// Mitsubishi GX Works2 project: PLC_GROUP15   PLC: FX3G

// global labels: Global1
VAR_GLOBAL
  startDay AT X007 : BOOL;
  stayOn AT Y007 : BOOL;
  analogOutput AT D8282 : INT;
  checkStock AT M1 : BOOL;
  theDayEnd AT M20 : BOOL;
  validStock AT M2 : BOOL;
  lifeDay AT Y007 : BOOL;
  helpDayStart AT M22 : BOOL;
  petelInput AT D1100 : REAL;
END_VAR
VAR_GLOBAL CONSTANT
  petelMin : REAL := 280;
END_VAR
VAR_GLOBAL
  limonInput AT D1200 : REAL;
END_VAR
VAR_GLOBAL CONSTANT
  limonMin : REAL := 455;
END_VAR
VAR_GLOBAL
  meiatzevInput AT D1300 : REAL;
END_VAR
VAR_GLOBAL CONSTANT
  meiatzevMin : REAL := 105;
END_VAR
VAR_GLOBAL
  gummiInput AT D1400 : REAL;
END_VAR
VAR_GLOBAL CONSTANT
  gummiMin : REAL := 28;
END_VAR
VAR_GLOBAL
  petelTotal AT D1102 : REAL;
  limonTotal AT D1202 : REAL;
  meiatzevTotal AT D1302 : REAL;
  gummiTotal AT D1402 : REAL;
  Dgima AT X001 : BOOL;
END_VAR
VAR_GLOBAL CONSTANT
  petelFor7Pinuk : REAL := 385;
  limonFor7Pinuk : REAL := 665;
  meiatzevFor7Pinuk : REAL := 210;
  gummiFor7Pinuk : REAL := 70;
END_VAR
VAR_GLOBAL
  checkPinukMlay AT M13 : BOOL;
  AnalogInput1 AT D8280 : INT;
END_VAR
VAR_GLOBAL CONSTANT
  Nirmul : REAL := 404.5;
END_VAR
VAR_GLOBAL
  iceCreamType AT D1502 : REAL;
END_VAR
VAR_GLOBAL CONSTANT
  minNormal : REAL;
  minimumPinuk : REAL := 6;
  maxNormal : REAL := 5.0;
END_VAR
VAR_GLOBAL
  checkMLAY AT M13 : BOOL;
  chooseNormal AT M3 : BOOL;
  choosePinuk AT M4 : BOOL;
  timerForMaking AT TC1 : BOOL;
END_VAR
VAR_GLOBAL CONSTANT
  secondsMaking : INT := 50;
END_VAR
VAR_GLOBAL
  endMaking AT TS1 : BOOL;
  onWhileMaking AT Y000 : BOOL;
END_VAR
VAR_GLOBAL CONSTANT
  meiatzevFor7NormalLemon : REAL := 70;
  meiatzevFor7NormalPetel : REAL := 35;
  meiatzevFor7PinukLemon : REAL := 140;
  meiatzevFor7PinukPetel : REAL := 70;
  limonFor7PinukLemon : REAL := 560;
  limonFor7PinukPetel : REAL := 105;
  limonFor7NormalLemon : REAL := 420;
  petelFor7NormalPetel : REAL := 280;
  petelFor7PinukPetel : REAL := 385;
  make7NormalLemon : REAL := 490;
END_VAR
VAR_GLOBAL
  limonBox AT D1800 : REAL;
END_VAR
VAR_GLOBAL CONSTANT
  make7Normalpetel : REAL := 350;
  make7PinukLimon : REAL := 700;
  make7PinukPetel : REAL := 560;
END_VAR
VAR_GLOBAL
  startFreezing AT X002 : BOOL;
  freezingLimon AT D1602 : REAL;
  onWhileFreezing AT Y002 : BOOL;
  freezingIcecream AT TC8 : BOOL;
END_VAR
VAR_GLOBAL CONSTANT
  freezingTime : INT := 80;
END_VAR
VAR_GLOBAL
  Bulb AT TS3 : BOOL;
  temp AT X003 : BOOL;
  ReadyToMix AT M0 : BOOL;
  ReadyToMix2 AT M30 : BOOL;
  DuringFreezing AT Y002 : BOOL;
END_VAR
VAR_GLOBAL CONSTANT
  lemonIceCreamForNormal : REAL := 490;
  petelIceCreamForNormal : REAL;
  gummiFor7Normal : REAL := 28;
END_VAR
VAR_GLOBAL
  MixingNormalTimer AT TC3 : BOOL;
END_VAR
VAR_GLOBAL CONSTANT
  MixingNormalTime : INT := 30;
END_VAR
VAR_GLOBAL
  HelpFlick AT M16 : BOOL;
  TC_4 AT TC4 : BOOL;
END_VAR
VAR_GLOBAL CONSTANT
  OnOf : INT := 20;
END_VAR
VAR_GLOBAL
  flickering AT Y005 : BOOL;
  flickering2 AT Y006 : BOOL;
  TS_5 AT TS5 : BOOL;
  TS_4 AT TS4 : BOOL;
  TC_5 AT TC5 : BOOL;
END_VAR
VAR_GLOBAL CONSTANT
  lemonIceCreamForPinuk : REAL := 700;
  petelIceCreamForPinuk : REAL := 560;
END_VAR
VAR_GLOBAL
  MixingPinukTimer AT TC5 : BOOL;
END_VAR
VAR_GLOBAL CONSTANT
  MixingPinukTime : INT := 50;
END_VAR
VAR_GLOBAL
  stopflicket AT Y005 : BOOL;
  stopflicker AT Y005 : BOOL;
  stopflicker2 AT Y006 : BOOL;
  startAriza AT X004 : BOOL;
  arizat1IceCream AT X000 : BOOL;
  countFirstIceCream AT CC0 : BOOL;
END_VAR
VAR_GLOBAL CONSTANT
  CounterFirstIcecream : INT := 1;
END_VAR
VAR_GLOBAL
  countPackage AT CC1 : BOOL;
END_VAR
VAR_GLOBAL CONSTANT
  counterPackages : INT := 7;
END_VAR
VAR_GLOBAL
  startCount AT CS0 : BOOL;
  finishCount AT CS1 : BOOL;
  startMore6 AT Y004 : BOOL;
  endOneIteration AT M10 : BOOL;
  Add7Icecream AT Y004 : BOOL;
  AddPackage AT Y004 : BOOL;
END_VAR
VAR_GLOBAL CONSTANT
  AddingPackage : REAL := 1;
END_VAR
VAR_GLOBAL
  endDay AT X005 : BOOL;
  MlayEndDay AT M12 : BOOL;
  endDayFINISH AT M5 : BOOL;
END_VAR
VAR_GLOBAL CONSTANT
  meiatzevFor7 : REAL := 70;
  petelFor7Normal : REAL := 280;
  limonFor7Normal : REAL := 455;
  meiatzevFor7Normal : REAL := 105;
  constant_40 : REAL := 40;
END_VAR
VAR_GLOBAL
  Output_package AT D1404 : REAL;
  TC_6 AT TC6 : BOOL;
  TS_6 AT TS6 : BOOL;
  petel_box AT D1700 : REAL;
  freezing_Petel AT D1702 : REAL;
  Normal_Box AT D1750 : REAL;
  pinuk_Box AT D1760 : REAL;
  Amount_Packages AT D1780 : REAL;
END_VAR
VAR_GLOBAL CONSTANT
  limonFor7PetelNormal : REAL := 35;
END_VAR

// task Task_01 (event TRUE, interval 0, priority 31): POU_01

PROGRAM POU_01
VAR CONSTANT
  nrtt : REAL;
END_VAR
(* structured ladder/FBD written out as ST: instructions are called as NAME(EN, inputs, outputs); _pN, _eN, _tN stand for wires *)
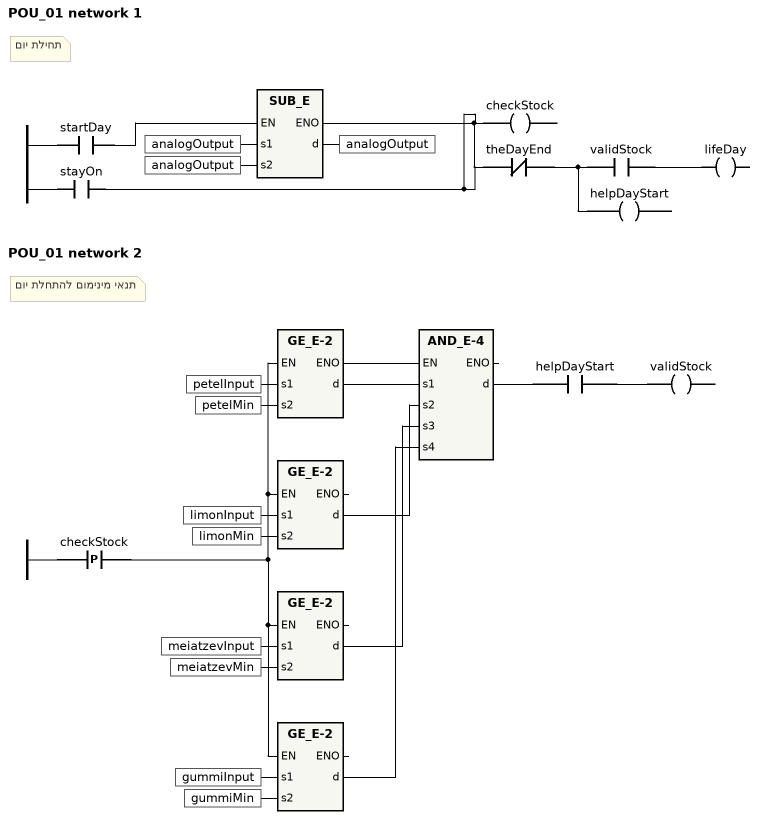
(* network 1 *)
(* תחילת יום *)
_e1 := SUB_E(startDay, analogOutput, analogOutput, analogOutput);
_p2 := _e1 OR stayOn;
checkStock := _p2;
_p3 := _p2 AND NOT theDayEnd;
lifeDay := _p3 AND validStock;
helpDayStart := _p3;
(* network 2 *)
(* תנאי מינימום להתחלת יום *)
_p1 := LDP(TRUE, checkStock);
_e3 := GE_E(_p1, petelInput, petelMin, _t2);
GE_E(_p1, limonInput, limonMin, _t4);
GE_E(_p1, meiatzevInput, meiatzevMin, _t5);
GE_E(_p1, gummiInput, gummiMin, _t6);
AND_E(_e3, _t2, _t4, _t5, _t6, _t7);
validStock := _t7 AND helpDayStart;
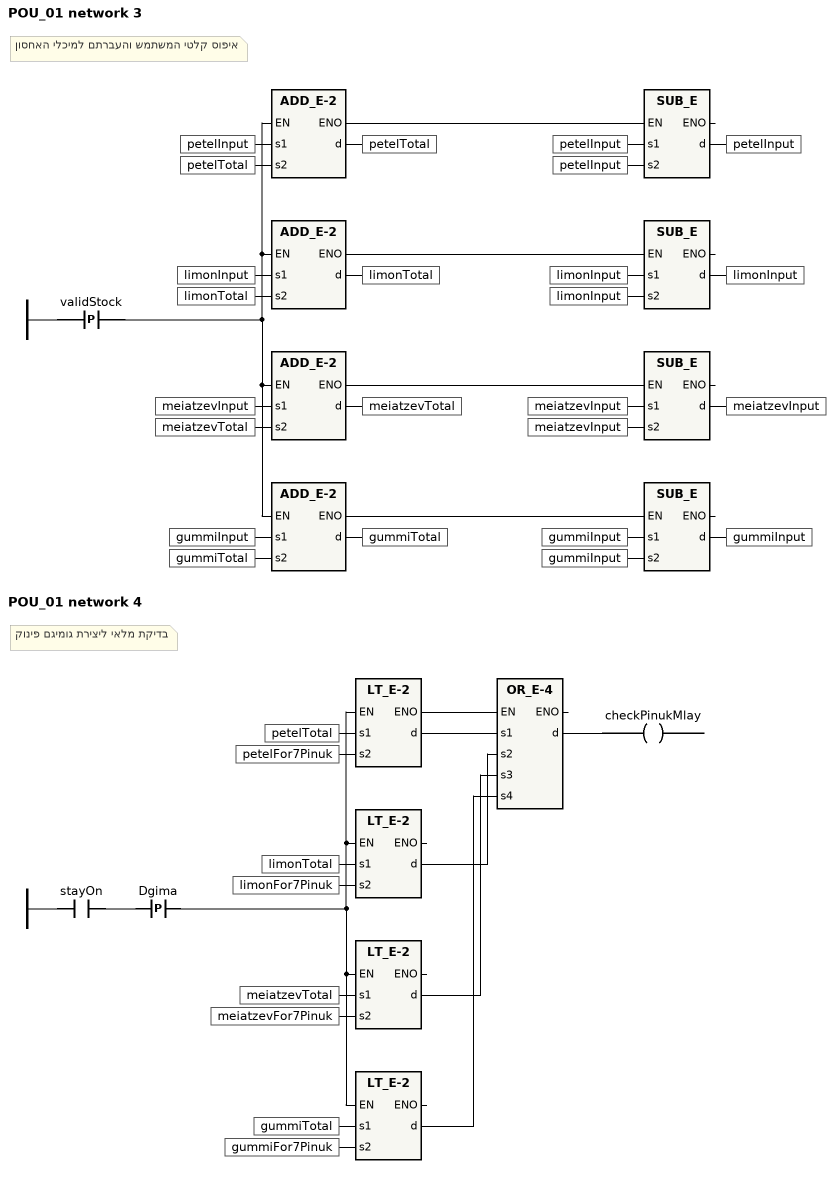
(* network 3 *)
(* איפוס קלטי המשתמש והעברתם למיכלי האחסון *)
_p1 := LDP(TRUE, validStock);
_e2 := ADD_E(_p1, petelInput, petelTotal, petelTotal);
SUB_E(_e2, petelInput, petelInput, petelInput);
_e3 := ADD_E(_p1, limonInput, limonTotal, limonTotal);
SUB_E(_e3, limonInput, limonInput, limonInput);
_e4 := ADD_E(_p1, meiatzevInput, meiatzevTotal, meiatzevTotal);
SUB_E(_e4, meiatzevInput, meiatzevInput, meiatzevInput);
_e5 := ADD_E(_p1, gummiInput, gummiTotal, gummiTotal);
SUB_E(_e5, gummiInput, gummiInput, gummiInput);
(* network 4 *)
(* בדיקת מלאי ליצירת גומיגם פינוק *)
_p1 := stayOn AND LDP(TRUE, Dgima);
_e3 := LT_E(_p1, petelTotal, petelFor7Pinuk, _t2);
LT_E(_p1, limonTotal, limonFor7Pinuk, _t4);
LT_E(_p1, meiatzevTotal, meiatzevFor7Pinuk, _t5);
LT_E(_p1, gummiTotal, gummiFor7Pinuk, _t6);
OR_E(_e3, _t2, _t4, _t5, _t6, _t7);
checkPinukMlay := _t7;
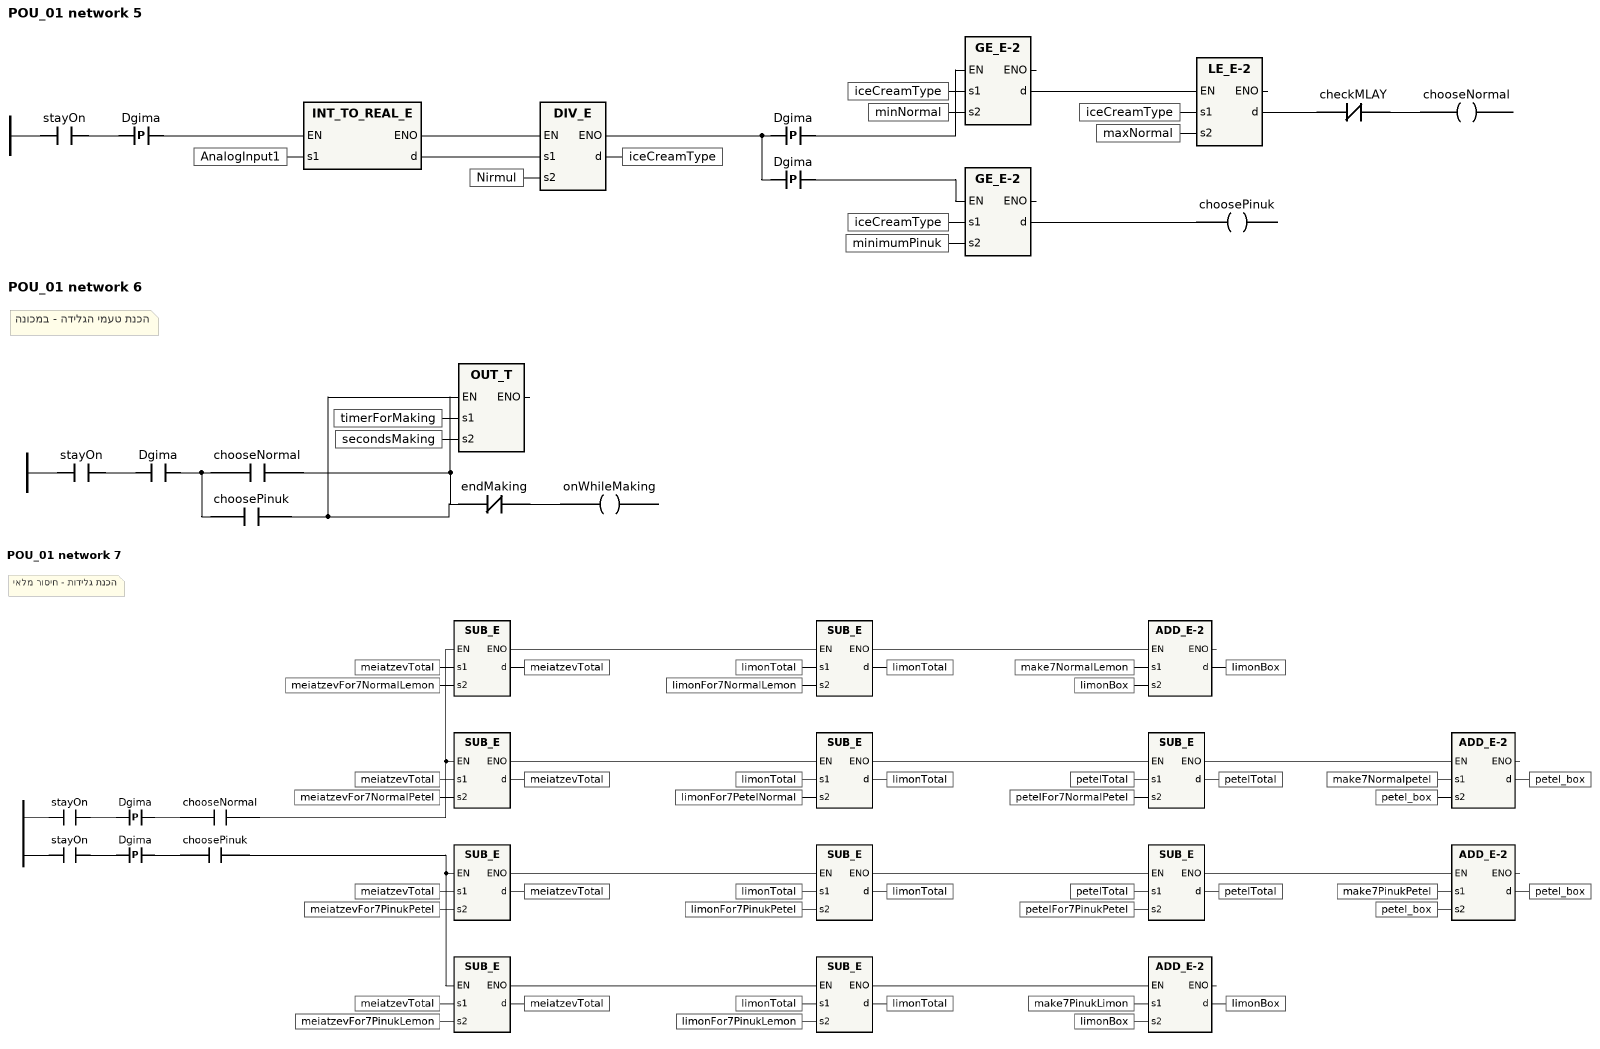
(* network 5 *)
_e2 := INT_TO_REAL_E(stayOn AND LDP(TRUE, Dgima), AnalogInput1, _t1);
_e3 := DIV_E(_e2, _t1, Nirmul, iceCreamType);
GE_E(_e3 AND LDP(TRUE, Dgima), iceCreamType, minNormal, _t4);
LE_E(_t4, iceCreamType, maxNormal, _t5);
chooseNormal := _t5 AND NOT checkMLAY;
GE_E(_e3 AND LDP(TRUE, Dgima), iceCreamType, minimumPinuk, _t6);
choosePinuk := _t6;
(* network 6 *)
(* הכנת טעמי הגלידה - במכונה *)
_p1 := stayOn AND Dgima;
_p2 := (_p1 AND chooseNormal) OR (_p1 AND choosePinuk);
OUT_T(_p2, timerForMaking, secondsMaking);
onWhileMaking := _p2 AND NOT endMaking;
(* network 7 *)
(* הכנת גלידות - חיסור מלאי *)
_p1 := stayOn AND LDP(TRUE, Dgima) AND chooseNormal;
_e2 := SUB_E(_p1, meiatzevTotal, meiatzevFor7NormalLemon, meiatzevTotal);
_e3 := SUB_E(_e2, limonTotal, limonFor7NormalLemon, limonTotal);
ADD_E(_e3, make7NormalLemon, limonBox, limonBox);
_e4 := SUB_E(_p1, meiatzevTotal, meiatzevFor7NormalPetel, meiatzevTotal);
_e5 := SUB_E(_e4, limonTotal, limonFor7PetelNormal, limonTotal);
_e6 := SUB_E(_e5, petelTotal, petelFor7NormalPetel, petelTotal);
ADD_E(_e6, make7Normalpetel, petel_box, petel_box);
_p7 := stayOn AND LDP(TRUE, Dgima) AND choosePinuk;
_e8 := SUB_E(_p7, meiatzevTotal, meiatzevFor7PinukLemon, meiatzevTotal);
_e9 := SUB_E(_e8, limonTotal, limonFor7PinukLemon, limonTotal);
ADD_E(_e9, make7PinukLimon, limonBox, limonBox);
_e10 := SUB_E(_p7, meiatzevTotal, meiatzevFor7PinukPetel, meiatzevTotal);
_e11 := SUB_E(_e10, limonTotal, limonFor7PinukPetel, limonTotal);
_e12 := SUB_E(_e11, petelTotal, petelFor7PinukPetel, petelTotal);
ADD_E(_e12, make7PinukPetel, petel_box, petel_box);
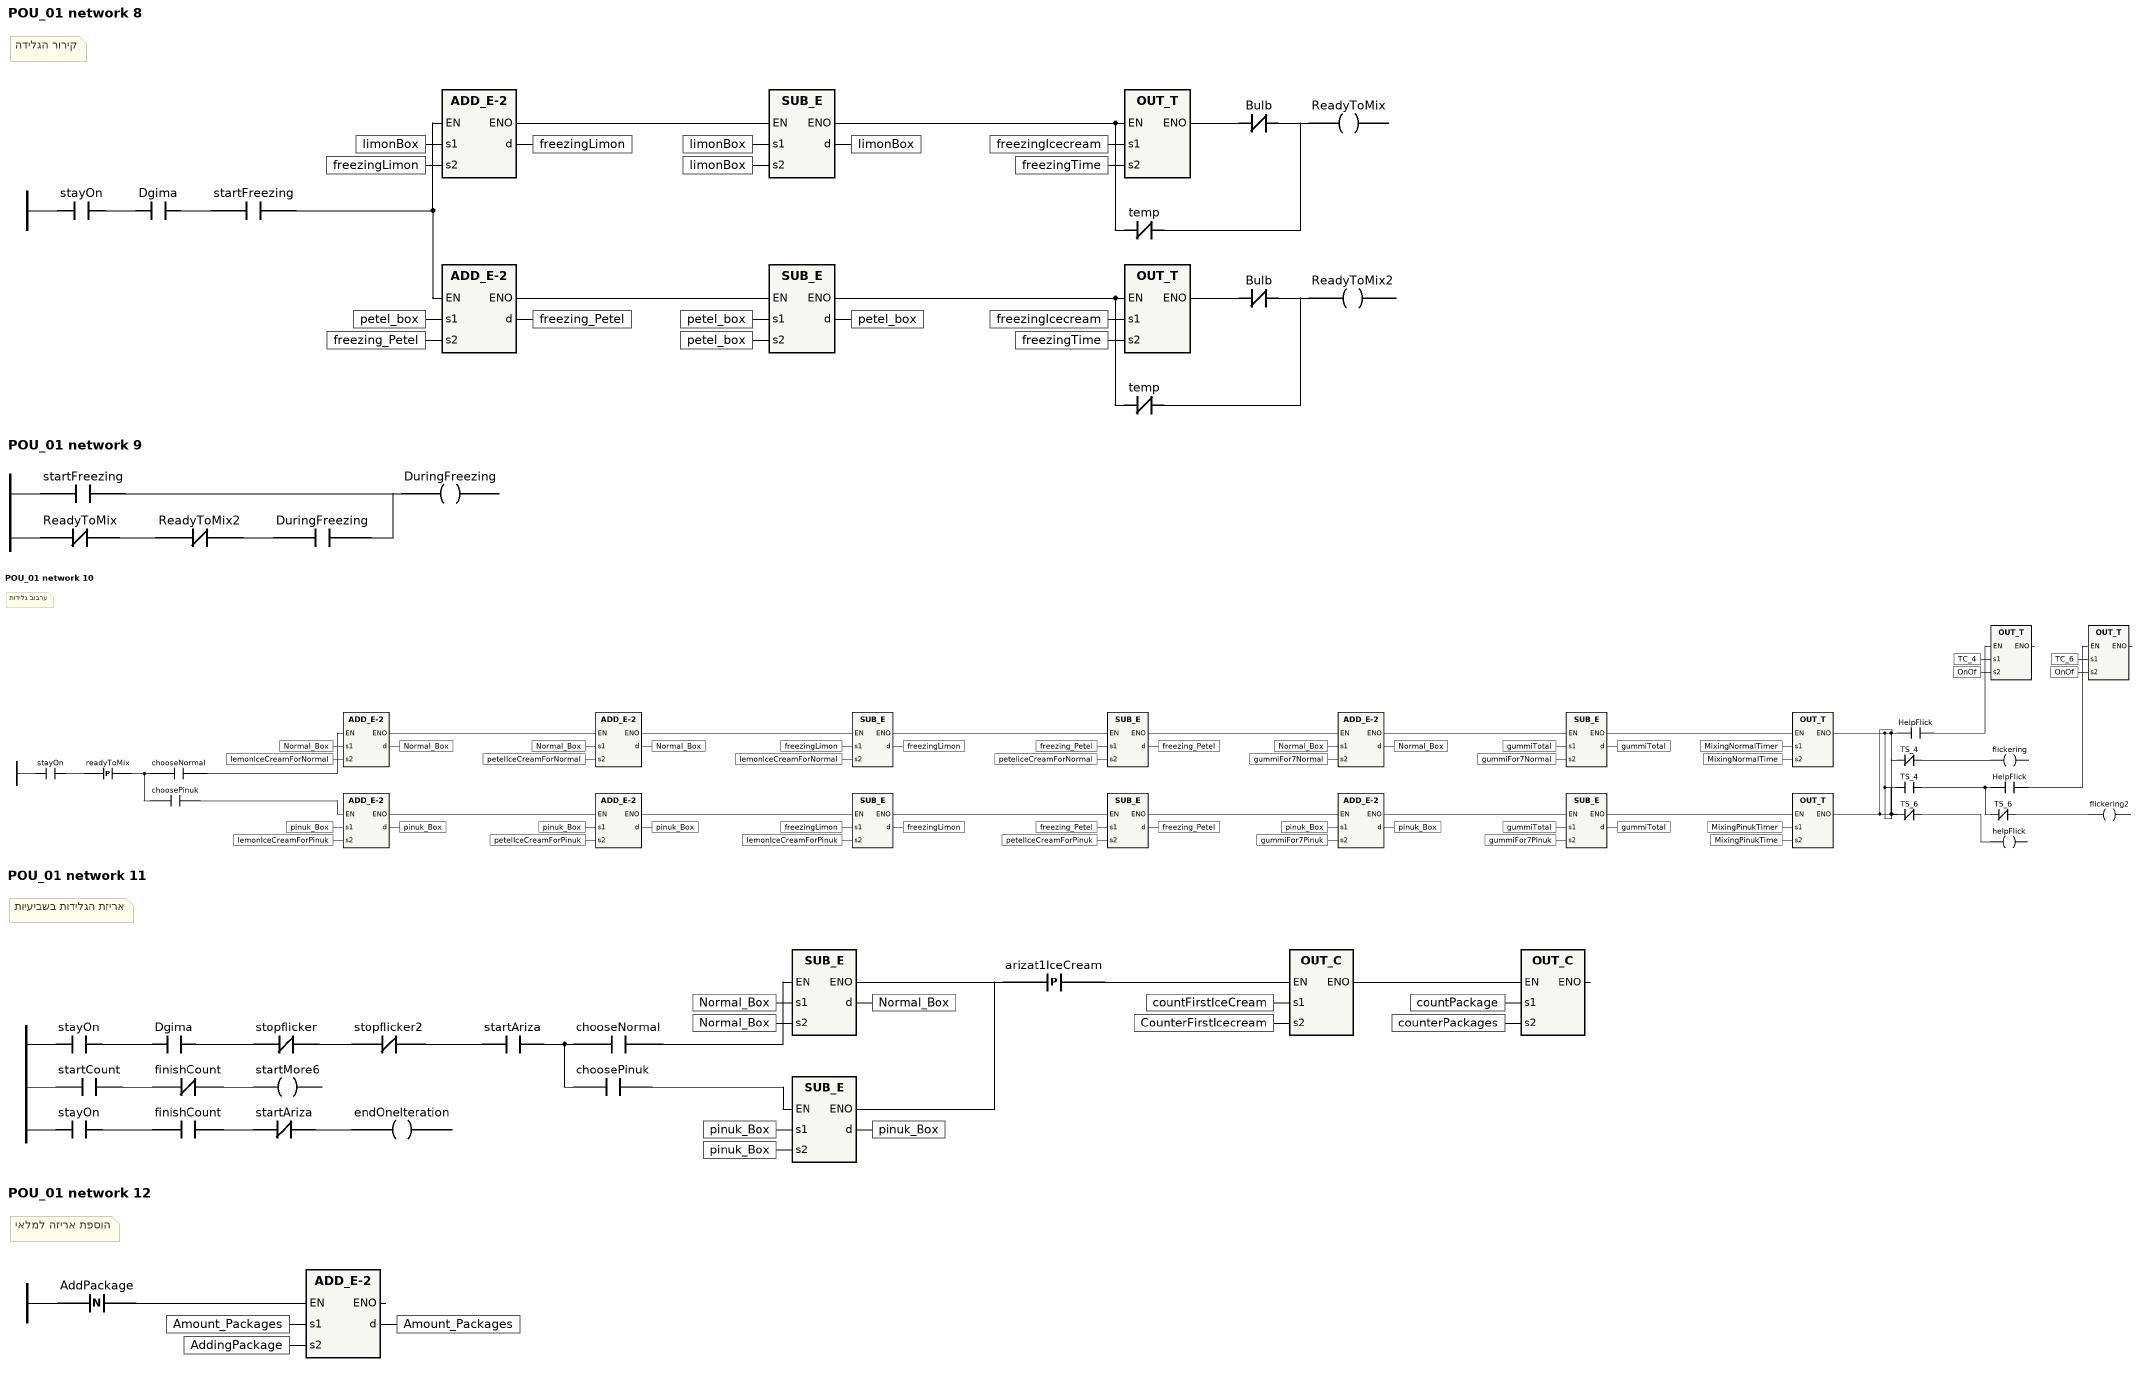
(* network 8 *)
(* קירור הגלידה *)
_p1 := stayOn AND Dgima AND startFreezing;
_e2 := ADD_E(_p1, limonBox, freezingLimon, freezingLimon);
_e3 := SUB_E(_e2, limonBox, limonBox, limonBox);
_e4 := OUT_T(_e3, freezingIcecream, freezingTime);
ReadyToMix := (_e4 AND NOT Bulb) OR (_e3 AND NOT temp);
_e5 := ADD_E(_p1, petel_box, freezing_Petel, freezing_Petel);
_e6 := SUB_E(_e5, petel_box, petel_box, petel_box);
_e7 := OUT_T(_e6, freezingIcecream, freezingTime);
ReadyToMix2 := (_e7 AND NOT Bulb) OR (_e6 AND NOT temp);
(* network 9 *)
DuringFreezing := startFreezing OR (NOT ReadyToMix AND NOT ReadyToMix2 AND DuringFreezing);
(* network 10 *)
(* ערבוב גלידות *)
_p1 := stayOn AND LDP(TRUE, readyToMix);
_e2 := ADD_E(_p1 AND chooseNormal, Normal_Box, lemonIceCreamForNormal, Normal_Box);
_e3 := ADD_E(_e2, Normal_Box, petelIceCreamForNormal, Normal_Box);
_e4 := SUB_E(_e3, freezingLimon, lemonIceCreamForNormal, freezingLimon);
_e5 := SUB_E(_e4, freezing_Petel, peteliceCreamForNormal, freezing_Petel);
_e6 := ADD_E(_e5, Normal_Box, gummiFor7Normal, Normal_Box);
_e7 := SUB_E(_e6, gummiTotal, gummiFor7Normal, gummiTotal);
_e8 := OUT_T(_e7, MixingNormalTimer, MixingNormalTime);
_e9 := ADD_E(_p1 AND choosePinuk, pinuk_Box, lemonIceCreamForPinuk, pinuk_Box);
_e10 := ADD_E(_e9, pinuk_Box, petelIceCreamForPinuk, pinuk_Box);
_e11 := SUB_E(_e10, freezingLimon, lemonIceCreamForPinuk, freezingLimon);
_e12 := SUB_E(_e11, freezing_Petel, petelIceCreamForPinuk, freezing_Petel);
_e13 := ADD_E(_e12, pinuk_Box, gummiFor7Pinuk, pinuk_Box);
_e14 := SUB_E(_e13, gummiTotal, gummiFor7Pinuk, gummiTotal);
_e15 := OUT_T(_e14, MixingPinukTimer, MixingPinukTime);
_p16 := _e8 OR _e15;
OUT_T(_p16 AND HelpFlick, TC_4, OnOf);
flickering := _p16 AND NOT TS_4;
_p17 := _p16 AND TS_4;
OUT_T(_p17 AND HelpFlick, TC_6, OnOf);
flickering2 := _p17 AND NOT TS_6;
helpFlick := _p16 AND NOT TS_6;
(* network 11 *)
(* אריזת הגלידות בשביעיות *)
_p1 := stayOn AND Dgima AND NOT stopflicker AND NOT stopflicker2 AND startAriza;
_e2 := SUB_E(_p1 AND chooseNormal, Normal_Box, Normal_Box, Normal_Box);
_e3 := SUB_E(_p1 AND choosePinuk, pinuk_Box, pinuk_Box, pinuk_Box);
_e4 := OUT_C((_e2 OR _e3) AND LDP(TRUE, arizat1IceCream), countFirstIceCream, CounterFirstIcecream);
OUT_C(_e4, countPackage, counterPackages);
startMore6 := startCount AND NOT finishCount;
endOneIteration := stayOn AND finishCount AND NOT startAriza;
(* network 12 *)
(* הוספת אריזה למלאי *)
ADD_E(LDF(TRUE, AddPackage), Amount_Packages, AddingPackage, Amount_Packages);
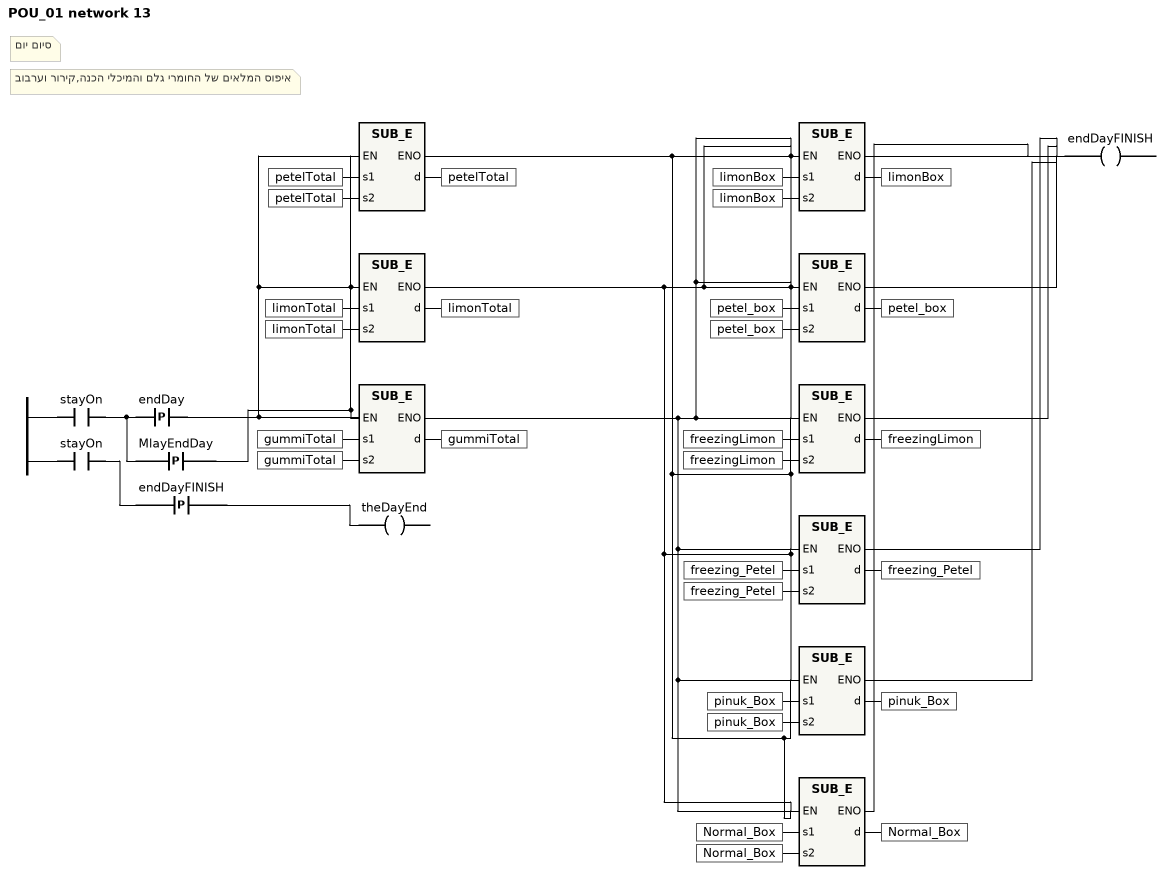
(* network 13 *)
(* סיום יום *)
(* איפוס המלאים של החומרי גלם והמיכלי הכנה,קירור וערבוב *)
_p1 := (stayOn AND LDP(TRUE, endDay)) OR (stayOn AND LDP(TRUE, MlayEndDay));
_e2 := SUB_E(_p1, petelTotal, petelTotal, petelTotal);
_e3 := SUB_E(_p1, limonTotal, limonTotal, limonTotal);
_e4 := SUB_E(_p1, gummiTotal, gummiTotal, gummiTotal);
_p5 := _e2 OR _e3 OR _e4;
_e6 := SUB_E(_p5, limonBox, limonBox, limonBox);
_e7 := SUB_E(_p5, petel_box, petel_box, petel_box);
_e8 := SUB_E(_p5, freezingLimon, freezingLimon, freezingLimon);
_e9 := SUB_E(_p5, freezing_Petel, freezing_Petel, freezing_Petel);
_e10 := SUB_E(_p5, pinuk_Box, pinuk_Box, pinuk_Box);
_e11 := SUB_E(_p5, Normal_Box, Normal_Box, Normal_Box);
endDayFINISH := _e6 OR _e7 OR _e8 OR _e9 OR _e10 OR _e11;
theDayEnd := stayOn AND LDP(TRUE, endDayFINISH);
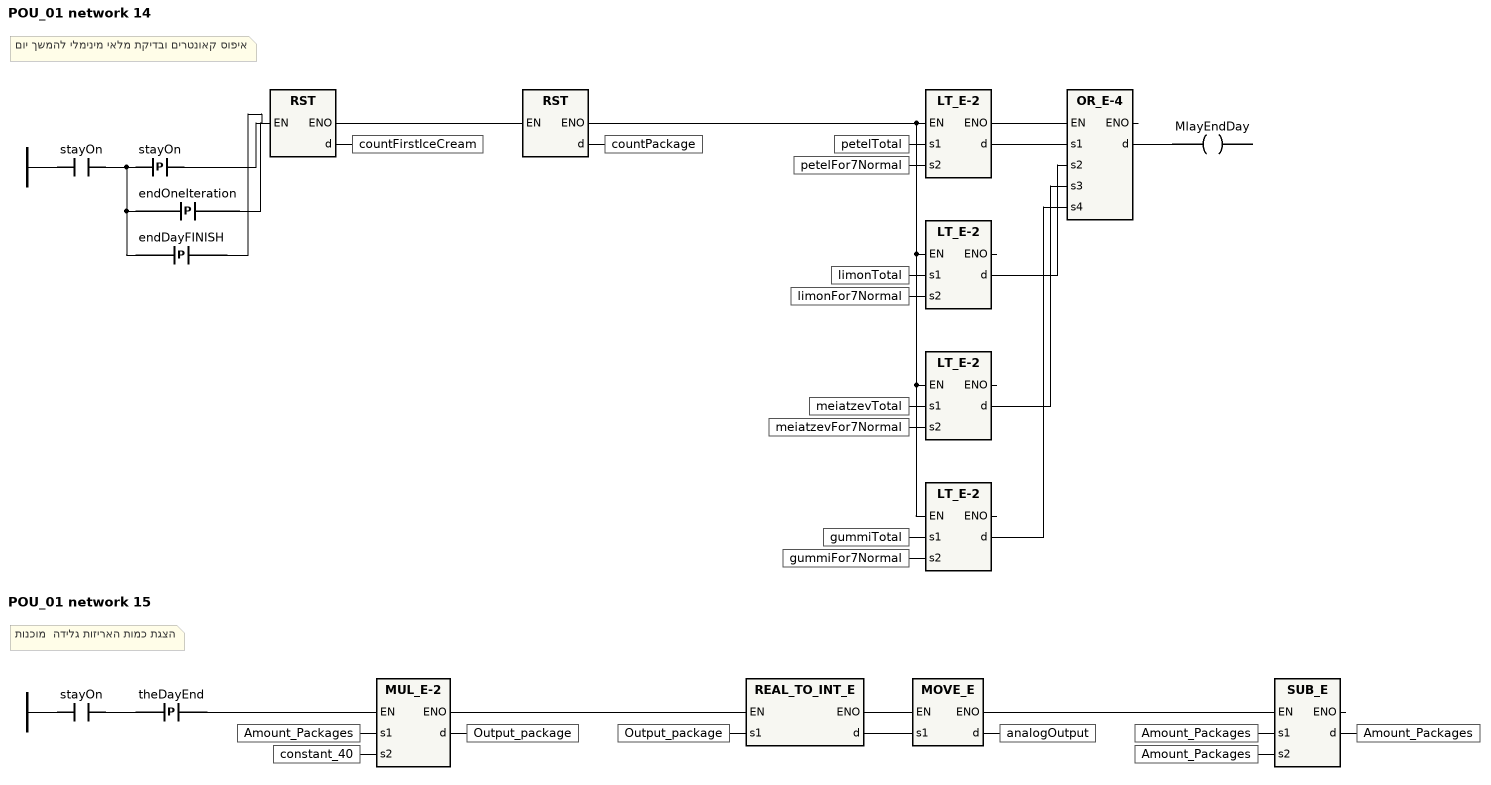
(* network 14 *)
(* איפוס קאונטרים ובדיקת מלאי מינימלי להמשך יום *)
_e1 := RST((stayOn AND LDP(TRUE, stayOn)) OR (stayOn AND LDP(TRUE, endOneIteration)) OR (stayOn AND LDP(TRUE, endDayFINISH)), countFirstIceCream);
_e2 := RST(_e1, countPackage);
_e4 := LT_E(_e2, petelTotal, petelFor7Normal, _t3);
LT_E(_e2, limonTotal, limonFor7Normal, _t5);
LT_E(_e2, meiatzevTotal, meiatzevFor7Normal, _t6);
LT_E(_e2, gummiTotal, gummiFor7Normal, _t7);
OR_E(_e4, _t3, _t5, _t6, _t7, _t8);
MlayEndDay := _t8;
(* network 15 *)
(* הצגת כמות האריזות גלידה  מוכנות *)
_e1 := MUL_E(stayOn AND LDP(TRUE, theDayEnd), Amount_Packages, constant_40, Output_package);
_e3 := REAL_TO_INT_E(_e1, Output_package, _t2);
_e4 := MOVE_E(_e3, _t2, analogOutput);
SUB_E(_e4, Amount_Packages, Amount_Packages, Amount_Packages);
END_PROGRAM
